{attribute 'GeneratedUsingTerminal: EK1100-0000-0018'}
{attribute addProperty BoxType "EK1100-0000-0018"}
{attribute addProperty Id "Beckhoff_ELM31xxEK1122Beckhoff_ELM31xxEK1122_DD4955802A_0001_ELM3102_0000_0016ELM3102_3D4ED79F42A_0002_ELM3102_0000_0017ELM3102_3D4ED79F42A_0003_ELM3102_0000_0018ELM3102_3D4ED79F42A_0004_ELM3104_0000_0016ELM3104_177D76D464A_0005_ELM3104_0000_0017ELM3104_177D76D464A_0006_ELM3104_0000_0018ELM3104_177D76D464A_0007_ELM3142_0000_0016ELM3142_3D4ED79F42A_0008_ELM3142_0000_0017ELM3142_3D4ED79F42A_0009_ELM3144_0000_0016ELM3144_177D76D464A_0010_ELM3144_0000_0017ELM3144_177D76D464A_0011_ELM3146_0000_0016ELM3146_6335DDA786A_0012_ELM3146_0000_0017ELM3146_6335DDA786A_0013_ELM3146_0000_0018ELM3146_6335DDA786A_0014_ELM3148_0000_0017ELM3148_8160AE58108A_0015_ELM3148_0000_0018ELM3148_8160AE58108A_0016_ELM3148_0000_0019ELM3148_8160AE58108"}
{attribute addProperty CRC "1812589244"}
{attribute addProperty Size "1114"}
TYPE Beckhoff_ELM31xx_6C09EABC EXTENDS EK1100_1FC0878B :
STRUCT
	{attribute addProperty Name "Beckhoff_ELM31xxEK1122"}
	{attribute addProperty PreviousPort "Beckhoff ELM31xx : B"}
	Beckhoff_ELM31xxEK1122 : Beckhoff_ELM31xxEK1122_DD495580;
	{attribute addProperty Name "A_0001_ELM3102_0000_0016"}
	{attribute addProperty PreviousPort "Beckhoff ELM31xxEK1122 : C"}
	A_0001_ELM3102_0000_0016 : ELM3102_3D4ED79F;
	{attribute addProperty Name "A_0002_ELM3102_0000_0017"}
	{attribute addProperty PreviousPort "A_0001(ELM3102-0000-0016) : B"}
	A_0002_ELM3102_0000_0017 : ELM3102_3D4ED79F;
	{attribute addProperty Name "A_0003_ELM3102_0000_0018"}
	{attribute addProperty PreviousPort "A_0002(ELM3102-0000-0017) : B"}
	A_0003_ELM3102_0000_0018 : ELM3102_3D4ED79F;
	{attribute addProperty Name "A_0004_ELM3104_0000_0016"}
	{attribute addProperty PreviousPort "A_0003(ELM3102-0000-0018) : B"}
	A_0004_ELM3104_0000_0016 : ELM3104_177D76D4;
	{attribute addProperty Name "A_0005_ELM3104_0000_0017"}
	{attribute addProperty PreviousPort "A_0004(ELM3104-0000-0016) : B"}
	A_0005_ELM3104_0000_0017 : ELM3104_177D76D4;
	{attribute addProperty Name "A_0006_ELM3104_0000_0018"}
	{attribute addProperty PreviousPort "A_0005(ELM3104-0000-0017) : B"}
	A_0006_ELM3104_0000_0018 : ELM3104_177D76D4;
	{attribute addProperty Name "A_0007_ELM3142_0000_0016"}
	{attribute addProperty PreviousPort "A_0006(ELM3104-0000-0018) : B"}
	A_0007_ELM3142_0000_0016 : ELM3142_3D4ED79F;
	{attribute addProperty Name "A_0008_ELM3142_0000_0017"}
	{attribute addProperty PreviousPort "A_0007(ELM3142-0000-0016) : B"}
	A_0008_ELM3142_0000_0017 : ELM3142_3D4ED79F;
	{attribute addProperty Name "A_0009_ELM3144_0000_0016"}
	{attribute addProperty PreviousPort "A_0008(ELM3142-0000-0017) : B"}
	A_0009_ELM3144_0000_0016 : ELM3144_177D76D4;
	{attribute addProperty Name "A_0010_ELM3144_0000_0017"}
	{attribute addProperty PreviousPort "A_0009(ELM3144-0000-0016) : B"}
	A_0010_ELM3144_0000_0017 : ELM3144_177D76D4;
	{attribute addProperty Name "A_0011_ELM3146_0000_0016"}
	{attribute addProperty PreviousPort "A_0010(ELM3144-0000-0017) : B"}
	A_0011_ELM3146_0000_0016 : ELM3146_6335DDA7;
	{attribute addProperty Name "A_0012_ELM3146_0000_0017"}
	{attribute addProperty PreviousPort "A_0011(ELM3146-0000-0016) : B"}
	A_0012_ELM3146_0000_0017 : ELM3146_6335DDA7;
	{attribute addProperty Name "A_0013_ELM3146_0000_0018"}
	{attribute addProperty PreviousPort "A_0012(ELM3146-0000-0017) : B"}
	A_0013_ELM3146_0000_0018 : ELM3146_6335DDA7;
	{attribute addProperty Name "A_0014_ELM3148_0000_0017"}
	{attribute addProperty PreviousPort "A_0013(ELM3146-0000-0018) : B"}
	A_0014_ELM3148_0000_0017 : ELM3148_8160AE58;
	{attribute addProperty Name "A_0015_ELM3148_0000_0018"}
	{attribute addProperty PreviousPort "A_0014(ELM3148-0000-0017) : B"}
	A_0015_ELM3148_0000_0018 : ELM3148_8160AE58;
	{attribute addProperty Name "A_0016_ELM3148_0000_0019"}
	{attribute addProperty PreviousPort "A_0015(ELM3148-0000-0018) : B"}
	A_0016_ELM3148_0000_0019 : ELM3148_8160AE58;
END_STRUCT
END_TYPE

(* stored: Version 1.2.0.0, ProductVersion 3.1.4024.9
   DUT Beckhoff_ELM31xx_6C09EABC: Id {6388dcf8-d7a5-4197-bf88-6a37119e1318} *)
